// Brief: Master Arm Standby
FUNCTION_BLOCK PUBLIC FB_StateCtrlStandBy EXTENDS FB_MasterArmCtrlBase
VAR_INPUT
END_VAR
VAR_OUTPUT
END_VAR
VAR
END_VAR

METHOD PUBLIC init : BOOL
VAR_IN_OUT CONSTANT
	i_masterArm	:FB_MasterArm;
END_VAR
VAR_IN_OUT 
	r_masterArmCtrlCmd :ST_ArmCtrlCmds;
END_VAR
// check if to hold the command joint position unchanged
m_holdLastCmds := checkToHoldLastCmds(i_masterArm);

// init
SUPER^.Init(i_masterArm,r_masterArmCtrlCmd);
END_METHOD

END_FUNCTION_BLOCK

(* stored: Version 1.1.0.1, ProductVersion 3.1.4024.11
   POU FB_StateCtrlStandBy: Id {82e389e4-7a38-4619-a14b-0246d1236311}, SpecialFunc None
   Method init: Id {e4eba8ef-1092-44ea-8fed-edb6d236e75a} *)
